// TIA Portal V20 export
DATA_BLOCK "dStruct_Axis"   // DB30140
{ S7_Optimized_Access := 'TRUE' }
// stored: AutoNumber false, MemoryReserve 100
   VAR
      gs_Axis { S7_SetPoint := 'True'} : Array[0..9] of "sAxis";
      gs_Axis_HMI_Init { S7_SetPoint := 'True'} : "sAxis_HMI";
   END_VAR
BEGIN
END_DATA_BLOCK
